// TIA Portal V20 export
TYPE "UDT_typePoint5"
   STRUCT
      x : LReal;   // Cartesian X position [mm]
      y : LReal;   // Cartesian Y position [mm]
      z : LReal;   // Cartesian Z position [mm]
      "a" : LReal;   // Wrist orientation rotation A [deg]
   END_STRUCT;
END_TYPE
